(* IEC 61131-3 sources: CODESYS-IO-Visualization/CODESYS-IO-Visualization.fbsproj/Pi.device.xml.v3^/Plc Logic.plclogic.xml.v3^/Application.application.xml.v3^/Programs/1_IO, 2 files *)

(* ---- IO_MapTagData.prg.st ---- *)
PROGRAM IO_MapTagData
VAR
END_VAR

// ********** Tag Mapping to IO **********

// Ambient Temperature: Site.Plant.AmbientTemp -> Slot 0, Channel 0
MapInstAFromIO(Data := Site.Plant.AmbientTemp, IO := IO.Rack_01.Modules[0].Channels[0]);

// Pump 1 Temperature: Site.Plant.Pump1.Temp -> Slot 0, Channel 1
MapInstAFromIO(Data := Site.Plant.Pump1.Temp, IO := IO.Rack_01.Modules[0].Channels[1]);

// Pump 1 Flow: Site.Plant.Pump1.Flow -> Slot 0, Channel 3
MapInstAFromIO(Data := Site.Plant.Pump1.Flow, IO := IO.Rack_01.Modules[0].Channels[3]);

// Pump 1 Inlet Valve: Site.Plant.Pump1.InletValve -> Pump_Inlet_Valve: 192.168.160.39
MapValveEquipFromRotork(Valve := Site.Plant.Pump1.InletValve, MB := Pump_Inlet_Valve_MB);

// Pump 1 Outlet Valve: Site.Plant.Pump1.OutletValve -> Pump_Outlet_Valve: 192.168.160.39
MapValveEquipFromRotork(Valve := Site.Plant.Pump1.OutletValve, MB := Pump_Outlet_Valve_MB);

// Pump 1 VFD: Site.Plant.Pump1.VFD
Site.Plant.Pump1.VFD.Raw.BOOL0[0] := IO.Rack_01.Modules[0].Channels[4].ValueDig;	// Running
Site.Plant.Pump1.VFD.Raw.BOOL0[1] := IO.Rack_01.Modules[0].Channels[5].ValueDig;	// VFD Fault
Site.Plant.Pump1.VFD.Raw.REAL0[0] := IO.Rack_01.Modules[0].Channels[2].ValueEu;	// VFD Speed
IO.Rack_01.Modules[0].Channels[6].ValueEu := Site.Plant.Pump1.VFD.Raw.REAL0[20];	// VFD Speed Cmd

IO.Rack_01.Modules[0].Channels[7].ValueEu := Site.Plant.Pump1.Flow.CurVal.Value;	// VFD Flow Output
IO.Rack_01.Modules[0].Channels[8].ValueDig := Site.Plant.Pump1.VFD.Running;	// VFD Running
IO.Rack_01.Modules[0].Channels[9].ValueDig := Site.Plant.Pump1.VFD.Failure[0].Active;	// VFD Failed

(* ---- Main_IO.prg.st ---- *)
PROGRAM Main_IO

VAR_INPUT
	Init: BOOL := TRUE;
END_VAR

// ****************** Hardware IO Processing ******************
CodeSysCPU(cpu := CPU);

// Assign Pointers for Rack and Modules
IF (Init) THEN
	Initialize();
END_IF;

SetRackIO();

// Set Rack and Module Status from hardware
Rack_Opto_RIO(Rack := Rack_01);

// Process all IO for Rack
ProcessRackIO_Opto(Rack := Rack_01);		// Process I/O to set values / status codes

// ****************** Fieldbus Device Processing ******************

// Valve 1 - 192.168.160.39 Port 502
Pump_Inlet_Valve_In.State := Pump_Inlet_Valve_Slave.ComState;
Pump_Inlet_Valve_In.Error := Pump_Inlet_Valve_Slave.xError;
Pump_Inlet_Valve_In.ErrorCode := Pump_Inlet_Valve_Slave.byModbusError;

RotorkValve(
	Data := Pump_Inlet_Valve_MB,
	InputData := Pump_Inlet_Valve_In,
	OutputData := Pump_Inlet_Valve_Out
);

// Valve 2 - 192.168.160.39 Port 503
Pump_Outlet_Valve_In.State := Pump_Outlet_Valve_Slave.ComState;
Pump_Outlet_Valve_In.Error := Pump_Outlet_Valve_Slave.xError;
Pump_Outlet_Valve_In.ErrorCode := Pump_Outlet_Valve_Slave.byModbusError;

RotorkValve(
	Data := Pump_Outlet_Valve_MB,
	InputData := Pump_Outlet_Valve_In,
	OutputData := Pump_Outlet_Valve_Out
);

// Map IO Points to Equipment and Instruments
IO_MapTagData();
